KUKA KRL program: UP999.src, Up999.dat

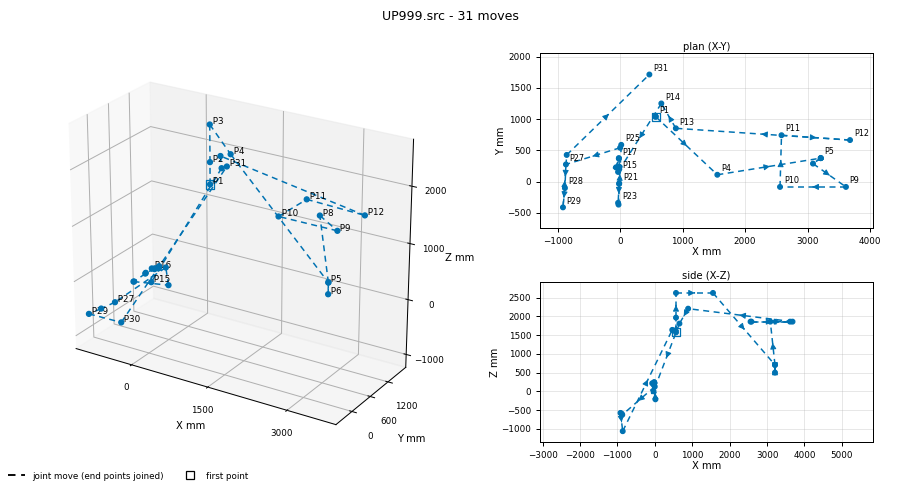
[picture p0: tool path of UP999.src, 31 of 31 moves have a stored position in this frame; points joined in program order, loops and branches not executed]
--- UP999.src ---
&ACCESS RVP2
&REL 75
&COMMENT israbiaoding
&PARAM EDITMASK = Up999[1-999]
&PARAM TPVW_VERSION = 8.3.17
&PARAM TEMPLATE = C:\KRC\Roboter\Template\upvorgabe
&PARAM DISKPATH = KRC:\R1\UPs
DEF UP999()
   ; FOLD UP Anfang;%{SE} %MKUKATPVW
   SPS_N=-1
   SPS_FERTIG=FALSE
   IF NOT CALLBYSELECT THEN
      INTERRUPT DECL 10 WHEN $CYCFLAG[254]==FALSE DO VW(#FB_STOP,TRUE)
      INTERRUPT ON 10
      INT10=TRUE
      VW_USR_R (#USR_INIT)
   ENDIF
   VW(#VW_INIT_UP,TRUE)
   ; ENDFOLD
   ;FOLD PTP VB=100% VE=0% ACC=100% RobWzg=0 Base=0 SPSTrig=0[1/100s]  ;%{P}%MKUKATPVW,%CMOVE8,%VPTP,%P 1:1, 2: VB=, 3:100, 4:%, 5: VE=, 6:0, 7:%, 8: ACC=, 9:100, 10:%, 11: RobWzg=, 12:0, 13: Base=, 14:0, 15: SPSTrig=, 16:0, 17:[1/100s], 18: , 19:1, 20:-1, 21:-1
      ;FOLD 1: ;%{SE}%MKUKATPVW
      ;ENDFOLD
      ;FOLD {H}
         VW_MPARA_ACT=P1_D
         Act_P1 = P1
         Act_P2 = P1
         VW(#MPARA,TRUE)
         PTP P1
         $ADVANCE=1
      ;ENDFOLD
   ;ENDFOLD
   ;FOLD PTP VB=100% VE=0% ACC=100% RobWzg=0 Base=0 SPSTrig=0[1/100s]  ;%{P}%MKUKATPVW,%CMOVE8,%VPTP,%P 1:1, 2: VB=, 3:100, 4:%, 5: VE=, 6:0, 7:%, 8: ACC=, 9:100, 10:%, 11: RobWzg=, 12:0, 13: Base=, 14:0, 15: SPSTrig=, 16:0, 17:[1/100s], 18: , 19:2, 20:-1, 21:-1
      ;FOLD 1: ;%{SE}%MKUKATPVW
      ;ENDFOLD
      ;FOLD {H}
         VW_MPARA_ACT=P2_D
         Act_P1 = P2
         Act_P2 = P2
         VW(#MPARA,TRUE)
         PTP P2
         $ADVANCE=1
      ;ENDFOLD
   ;ENDFOLD
   ;FOLD PTP VB=100% VE=0% ACC=100% RobWzg=0 Base=0 SPSTrig=0[1/100s]  ;%{P}%MKUKATPVW,%CMOVE8,%VPTP,%P 1:1, 2: VB=, 3:100, 4:%, 5: VE=, 6:0, 7:%, 8: ACC=, 9:100, 10:%, 11: RobWzg=, 12:0, 13: Base=, 14:0, 15: SPSTrig=, 16:0, 17:[1/100s], 18: , 19:3, 20:-1, 21:-1
      ;FOLD 1: ;%{SE}%MKUKATPVW
      ;ENDFOLD
      ;FOLD {H}
         VW_MPARA_ACT=P3_D
         Act_P1 = P3
         Act_P2 = P3
         VW(#MPARA,TRUE)
         PTP P3
         $ADVANCE=1
      ;ENDFOLD
   ;ENDFOLD
   ;FOLD PTP VB=100% VE=0% ACC=100% RobWzg=0 Base=0 SPSTrig=0[1/100s]  ;%{P}%MKUKATPVW,%CMOVE8,%VPTP,%P 1:1, 2: VB=, 3:100, 4:%, 5: VE=, 6:0, 7:%, 8: ACC=, 9:100, 10:%, 11: RobWzg=, 12:0, 13: Base=, 14:0, 15: SPSTrig=, 16:0, 17:[1/100s], 18: , 19:4, 20:-1, 21:-1
      ;FOLD 1: ;%{SE}%MKUKATPVW
      ;ENDFOLD
      ;FOLD {H}
         VW_MPARA_ACT=P4_D
         Act_P1 = P4
         Act_P2 = P4
         VW(#MPARA,TRUE)
         PTP P4
         $ADVANCE=1
      ;ENDFOLD
   ;ENDFOLD
   ;FOLD PTP VB=100% VE=0% ACC=100% RobWzg=21 Base=0 SPSTrig=0[1/100s]  ;%{P}%MKUKATPVW,%CMOVE8,%VPTP,%P 1:1, 2: VB=, 3:100, 4:%, 5: VE=, 6:0, 7:%, 8: ACC=, 9:100, 10:%, 11: RobWzg=, 12:21, 13: Base=, 14:0, 15: SPSTrig=, 16:0, 17:[1/100s], 18: , 19:5, 20:-1, 21:-1
      ;FOLD 1: ;%{SE}%MKUKATPVW
      ;ENDFOLD
      ;FOLD {H}
         VW_MPARA_ACT=P5_D
         Act_P1 = P5
         Act_P2 = P5
         VW(#MPARA,TRUE)
         PTP P5
         $ADVANCE=1
      ;ENDFOLD
   ;ENDFOLD
   ;FOLD -- zhongxintcp -- ;%{PSE}%MKUKATPVW,%CVW_COM,%VCOMMENT,%P 1:Comment:, 2:zhongxintcp
      ;FOLD {H}
         M_COMMENT("zhongxintcp")
      ;ENDFOLD
   ;ENDFOLD
   ;FOLD PTP VB=100% VE=0% ACC=100% RobWzg=21 Base=0 SPSTrig=0[1/100s]  ;%{P}%MKUKATPVW,%CMOVE8,%VPTP,%P 1:1, 2: VB=, 3:100, 4:%, 5: VE=, 6:0, 7:%, 8: ACC=, 9:100, 10:%, 11: RobWzg=, 12:21, 13: Base=, 14:0, 15: SPSTrig=, 16:0, 17:[1/100s], 18: , 19:6, 20:-1, 21:-1
      ;FOLD 1: ;%{SE}%MKUKATPVW
      ;ENDFOLD
      ;FOLD {H}
         VW_MPARA_ACT=P6_D
         Act_P1 = P6
         Act_P2 = P6
         VW(#MPARA,TRUE)
         PTP P6
         $ADVANCE=1
      ;ENDFOLD
   ;ENDFOLD
   ;FOLD PTP VB=100% VE=0% ACC=100% RobWzg=21 Base=0 SPSTrig=0[1/100s]  ;%{P}%MKUKATPVW,%CMOVE8,%VPTP,%P 1:1, 2: VB=, 3:100, 4:%, 5: VE=, 6:0, 7:%, 8: ACC=, 9:100, 10:%, 11: RobWzg=, 12:21, 13: Base=, 14:0, 15: SPSTrig=, 16:0, 17:[1/100s], 18: , 19:7, 20:-1, 21:-1
      ;FOLD 1: ;%{SE}%MKUKATPVW
      ;ENDFOLD
      ;FOLD {H}
         VW_MPARA_ACT=P7_D
         Act_P1 = P7
         Act_P2 = P7
         VW(#MPARA,TRUE)
         PTP P7
         $ADVANCE=1
      ;ENDFOLD
   ;ENDFOLD
   ;FOLD -- 1zhong -- ;%{PSE}%MKUKATPVW,%CVW_COM,%VCOMMENT,%P 1:Comment:, 2:1zhong
      ;FOLD {H}
         M_COMMENT("1zhong")
      ;ENDFOLD
   ;ENDFOLD
   ;FOLD PTP VB=100% VE=0% ACC=100% RobWzg=0 Base=0 SPSTrig=0[1/100s]  ;%{P}%MKUKATPVW,%CMOVE8,%VPTP,%P 1:1, 2: VB=, 3:100, 4:%, 5: VE=, 6:0, 7:%, 8: ACC=, 9:100, 10:%, 11: RobWzg=, 12:0, 13: Base=, 14:0, 15: SPSTrig=, 16:0, 17:[1/100s], 18: , 19:8, 20:-1, 21:-1
      ;FOLD 1: ;%{SE}%MKUKATPVW
      ;ENDFOLD
      ;FOLD {H}
         VW_MPARA_ACT=P8_D
         Act_P1 = P8
         Act_P2 = P8
         VW(#MPARA,TRUE)
         PTP P8
         $ADVANCE=1
      ;ENDFOLD
   ;ENDFOLD
   ;FOLD -- 2 -- ;%{PSE}%MKUKATPVW,%CVW_COM,%VCOMMENT,%P 1:Comment:, 2:2
      ;FOLD {H}
         M_COMMENT("2")
      ;ENDFOLD
   ;ENDFOLD
   ;FOLD PTP VB=100% VE=0% ACC=100% RobWzg=0 Base=0 SPSTrig=0[1/100s]  ;%{P}%MKUKATPVW,%CMOVE8,%VPTP,%P 1:1, 2: VB=, 3:100, 4:%, 5: VE=, 6:0, 7:%, 8: ACC=, 9:100, 10:%, 11: RobWzg=, 12:0, 13: Base=, 14:0, 15: SPSTrig=, 16:0, 17:[1/100s], 18: , 19:9, 20:-1, 21:-1
      ;FOLD 1: ;%{SE}%MKUKATPVW
      ;ENDFOLD
      ;FOLD {H}
         VW_MPARA_ACT=P9_D
         Act_P1 = P9
         Act_P2 = P9
         VW(#MPARA,TRUE)
         PTP P9
         $ADVANCE=1
      ;ENDFOLD
   ;ENDFOLD
   ;FOLD -- 3 -- ;%{PSE}%MKUKATPVW,%CVW_COM,%VCOMMENT,%P 1:Comment:, 2:3
      ;FOLD {H}
         M_COMMENT("3")
      ;ENDFOLD
   ;ENDFOLD
   ;FOLD PTP VB=100% VE=0% ACC=100% RobWzg=0 Base=0 SPSTrig=0[1/100s]  ;%{P}%MKUKATPVW,%CMOVE8,%VPTP,%P 1:1, 2: VB=, 3:100, 4:%, 5: VE=, 6:0, 7:%, 8: ACC=, 9:100, 10:%, 11: RobWzg=, 12:0, 13: Base=, 14:0, 15: SPSTrig=, 16:0, 17:[1/100s], 18: , 19:10, 20:-1, 21:-1
      ;FOLD 1: ;%{SE}%MKUKATPVW
      ;ENDFOLD
      ;FOLD {H}
         VW_MPARA_ACT=P10_D
         Act_P1 = P10
         Act_P2 = P10
         VW(#MPARA,TRUE)
         PTP P10
         $ADVANCE=1
      ;ENDFOLD
   ;ENDFOLD
   ;FOLD -- 4 -- ;%{PSE}%MKUKATPVW,%CVW_COM,%VCOMMENT,%P 1:Comment:, 2:4
      ;FOLD {H}
         M_COMMENT("4")
      ;ENDFOLD
   ;ENDFOLD
   ;FOLD PTP VB=100% VE=0% ACC=100% RobWzg=0 Base=0 SPSTrig=0[1/100s]  ;%{P}%MKUKATPVW,%CMOVE8,%VPTP,%P 1:1, 2: VB=, 3:100, 4:%, 5: VE=, 6:0, 7:%, 8: ACC=, 9:100, 10:%, 11: RobWzg=, 12:0, 13: Base=, 14:0, 15: SPSTrig=, 16:0, 17:[1/100s], 18: , 19:11, 20:-1, 21:-1
      ;FOLD 1: ;%{SE}%MKUKATPVW
      ;ENDFOLD
      ;FOLD {H}
         VW_MPARA_ACT=P11_D
         Act_P1 = P11
         Act_P2 = P11
         VW(#MPARA,TRUE)
         PTP P11
         $ADVANCE=1
      ;ENDFOLD
   ;ENDFOLD
   ;FOLD -- 5 -- ;%{PSE}%MKUKATPVW,%CVW_COM,%VCOMMENT,%P 1:Comment:, 2:5
      ;FOLD {H}
         M_COMMENT("5")
      ;ENDFOLD
   ;ENDFOLD
   ;FOLD PTP VB=100% VE=0% ACC=100% RobWzg=0 Base=0 SPSTrig=0[1/100s]  ;%{P}%MKUKATPVW,%CMOVE8,%VPTP,%P 1:1, 2: VB=, 3:100, 4:%, 5: VE=, 6:0, 7:%, 8: ACC=, 9:100, 10:%, 11: RobWzg=, 12:0, 13: Base=, 14:0, 15: SPSTrig=, 16:0, 17:[1/100s], 18: , 19:12, 20:-1, 21:-1
      ;FOLD 1: ;%{SE}%MKUKATPVW
      ;ENDFOLD
      ;FOLD {H}
         VW_MPARA_ACT=P12_D
         Act_P1 = P12
         Act_P2 = P12
         VW(#MPARA,TRUE)
         PTP P12
         $ADVANCE=1
      ;ENDFOLD
   ;ENDFOLD
   ;FOLD -- redian -- ;%{PSE}%MKUKATPVW,%CVW_COM,%VCOMMENT,%P 1:Comment:, 2:redian
      ;FOLD {H}
         M_COMMENT("redian")
      ;ENDFOLD
   ;ENDFOLD
   ;FOLD PTP VB=100% VE=0% ACC=100% RobWzg=0 Base=0 SPSTrig=0[1/100s]  ;%{P}%MKUKATPVW,%CMOVE8,%VPTP,%P 1:1, 2: VB=, 3:100, 4:%, 5: VE=, 6:0, 7:%, 8: ACC=, 9:100, 10:%, 11: RobWzg=, 12:0, 13: Base=, 14:0, 15: SPSTrig=, 16:0, 17:[1/100s], 18: , 19:13, 20:-1, 21:-1
      ;FOLD 1: ;%{SE}%MKUKATPVW
      ;ENDFOLD
      ;FOLD {H}
         VW_MPARA_ACT=P13_D
         Act_P1 = P13
         Act_P2 = P13
         VW(#MPARA,TRUE)
         PTP P13
         $ADVANCE=1
      ;ENDFOLD
   ;ENDFOLD
   ;FOLD PTP VB=100% VE=0% ACC=100% RobWzg=0 Base=0 SPSTrig=0[1/100s]  ;%{P}%MKUKATPVW,%CMOVE8,%VPTP,%P 1:1, 2: VB=, 3:100, 4:%, 5: VE=, 6:0, 7:%, 8: ACC=, 9:100, 10:%, 11: RobWzg=, 12:0, 13: Base=, 14:0, 15: SPSTrig=, 16:0, 17:[1/100s], 18: , 19:14, 20:-1, 21:-1
      ;FOLD 1: ;%{SE}%MKUKATPVW
      ;ENDFOLD
      ;FOLD {H}
         VW_MPARA_ACT=P14_D
         Act_P1 = P14
         Act_P2 = P14
         VW(#MPARA,TRUE)
         PTP P14
         $ADVANCE=1
      ;ENDFOLD
   ;ENDFOLD
   ;FOLD PTP VB=100% VE=0% ACC=100% RobWzg=21 Base=21 SPSTrig=0[1/100s]  ;%{P}%MKUKATPVW,%CMOVE8,%VPTP,%P 1:1, 2: VB=, 3:100, 4:%, 5: VE=, 6:0, 7:%, 8: ACC=, 9:100, 10:%, 11: RobWzg=, 12:21, 13: Base=, 14:21, 15: SPSTrig=, 16:0, 17:[1/100s], 18: , 19:15, 20:-1, 21:-1
      ;FOLD 1: ;%{SE}%MKUKATPVW
      ;ENDFOLD
      ;FOLD {H}
         VW_MPARA_ACT=P15_D
         Act_P1 = P15
         Act_P2 = P15
         VW(#MPARA,TRUE)
         PTP P15
         $ADVANCE=1
      ;ENDFOLD
   ;ENDFOLD
   ;FOLD PTP VB=100% VE=0% ACC=100% RobWzg=21 Base=21 SPSTrig=0[1/100s]  ;%{P}%MKUKATPVW,%CMOVE8,%VPTP,%P 1:1, 2: VB=, 3:100, 4:%, 5: VE=, 6:0, 7:%, 8: ACC=, 9:100, 10:%, 11: RobWzg=, 12:21, 13: Base=, 14:21, 15: SPSTrig=, 16:0, 17:[1/100s], 18: , 19:16, 20:-1, 21:-1
      ;FOLD 1: ;%{SE}%MKUKATPVW
      ;ENDFOLD
      ;FOLD {H}
         VW_MPARA_ACT=P16_D
         Act_P1 = P16
         Act_P2 = P16
         VW(#MPARA,TRUE)
         PTP P16
         $ADVANCE=1
      ;ENDFOLD
   ;ENDFOLD
   ;FOLD -- 1zs -- ;%{PSE}%MKUKATPVW,%CVW_COM,%VCOMMENT,%P 1:Comment:, 2:1zs
      ;FOLD {H}
         M_COMMENT("1zs")
      ;ENDFOLD
   ;ENDFOLD
   ;FOLD PTP VB=100% VE=0% ACC=100% RobWzg=21 Base=21 SPSTrig=0[1/100s]  ;%{P}%MKUKATPVW,%CMOVE8,%VPTP,%P 1:1, 2: VB=, 3:100, 4:%, 5: VE=, 6:0, 7:%, 8: ACC=, 9:100, 10:%, 11: RobWzg=, 12:21, 13: Base=, 14:21, 15: SPSTrig=, 16:0, 17:[1/100s], 18: , 19:17, 20:-1, 21:-1
      ;FOLD 1: ;%{SE}%MKUKATPVW
      ;ENDFOLD
      ;FOLD {H}
         VW_MPARA_ACT=P17_D
         Act_P1 = P17
         Act_P2 = P17
         VW(#MPARA,TRUE)
         PTP P17
         $ADVANCE=1
      ;ENDFOLD
   ;ENDFOLD
   ;FOLD PTP VB=100% VE=0% ACC=100% RobWzg=21 Base=21 SPSTrig=0[1/100s]  ;%{P}%MKUKATPVW,%CMOVE8,%VPTP,%P 1:1, 2: VB=, 3:100, 4:%, 5: VE=, 6:0, 7:%, 8: ACC=, 9:100, 10:%, 11: RobWzg=, 12:21, 13: Base=, 14:21, 15: SPSTrig=, 16:0, 17:[1/100s], 18: , 19:18, 20:-1, 21:-1
      ;FOLD 1: ;%{SE}%MKUKATPVW
      ;ENDFOLD
      ;FOLD {H}
         VW_MPARA_ACT=P18_D
         Act_P1 = P18
         Act_P2 = P18
         VW(#MPARA,TRUE)
         PTP P18
         $ADVANCE=1
      ;ENDFOLD
   ;ENDFOLD
   ;FOLD -- 2ys -- ;%{PSE}%MKUKATPVW,%CVW_COM,%VCOMMENT,%P 1:Comment:, 2:2ys
      ;FOLD {H}
         M_COMMENT("2ys")
      ;ENDFOLD
   ;ENDFOLD
   ;FOLD PTP VB=100% VE=0% ACC=100% RobWzg=21 Base=21 SPSTrig=0[1/100s]  ;%{P}%MKUKATPVW,%CMOVE8,%VPTP,%P 1:1, 2: VB=, 3:100, 4:%, 5: VE=, 6:0, 7:%, 8: ACC=, 9:100, 10:%, 11: RobWzg=, 12:21, 13: Base=, 14:21, 15: SPSTrig=, 16:0, 17:[1/100s], 18: , 19:19, 20:-1, 21:-1
      ;FOLD 1: ;%{SE}%MKUKATPVW
      ;ENDFOLD
      ;FOLD {H}
         VW_MPARA_ACT=P19_D
         Act_P1 = P19
         Act_P2 = P19
         VW(#MPARA,TRUE)
         PTP P19
         $ADVANCE=1
      ;ENDFOLD
   ;ENDFOLD
   ;FOLD PTP VB=100% VE=0% ACC=100% RobWzg=21 Base=21 SPSTrig=0[1/100s]  ;%{P}%MKUKATPVW,%CMOVE8,%VPTP,%P 1:1, 2: VB=, 3:100, 4:%, 5: VE=, 6:0, 7:%, 8: ACC=, 9:100, 10:%, 11: RobWzg=, 12:21, 13: Base=, 14:21, 15: SPSTrig=, 16:0, 17:[1/100s], 18: , 19:20, 20:-1, 21:-1
      ;FOLD 1: ;%{SE}%MKUKATPVW
      ;ENDFOLD
      ;FOLD {H}
         VW_MPARA_ACT=P20_D
         Act_P1 = P20
         Act_P2 = P20
         VW(#MPARA,TRUE)
         PTP P20
         $ADVANCE=1
      ;ENDFOLD
   ;ENDFOLD
   ;FOLD -- 3zx -- ;%{PSE}%MKUKATPVW,%CVW_COM,%VCOMMENT,%P 1:Comment:, 2:3zx
      ;FOLD {H}
         M_COMMENT("3zx")
      ;ENDFOLD
   ;ENDFOLD
   ;FOLD PTP VB=100% VE=0% ACC=100% RobWzg=21 Base=21 SPSTrig=0[1/100s]  ;%{P}%MKUKATPVW,%CMOVE8,%VPTP,%P 1:1, 2: VB=, 3:100, 4:%, 5: VE=, 6:0, 7:%, 8: ACC=, 9:100, 10:%, 11: RobWzg=, 12:21, 13: Base=, 14:21, 15: SPSTrig=, 16:0, 17:[1/100s], 18: , 19:21, 20:-1, 21:-1
      ;FOLD 1: ;%{SE}%MKUKATPVW
      ;ENDFOLD
      ;FOLD {H}
         VW_MPARA_ACT=P21_D
         Act_P1 = P21
         Act_P2 = P21
         VW(#MPARA,TRUE)
         PTP P21
         $ADVANCE=1
      ;ENDFOLD
   ;ENDFOLD
   ;FOLD PTP VB=100% VE=0% ACC=100% RobWzg=21 Base=21 SPSTrig=5[1/100s]  ;%{P}%MKUKATPVW,%CMOVE8,%VPTP,%P 1:1, 2: VB=, 3:100, 4:%, 5: VE=, 6:0, 7:%, 8: ACC=, 9:100, 10:%, 11: RobWzg=, 12:21, 13: Base=, 14:21, 15: SPSTrig=, 16:5, 17:[1/100s], 18: , 19:22, 20:-1, 21:-1
      ;FOLD 1: ;%{SE}%MKUKATPVW
      ;ENDFOLD
      ;FOLD {H}
         VW_MPARA_ACT=P22_D
         Act_P1 = P22
         Act_P2 = P22
         VW(#MPARA,TRUE)
         PTP P22
         $ADVANCE=1
      ;ENDFOLD
   ;ENDFOLD
   ;FOLD -- 4zz -- ;%{PSE}%MKUKATPVW,%CVW_COM,%VCOMMENT,%P 1:Comment:, 2:4zz
      ;FOLD {H}
         M_COMMENT("4zz")
      ;ENDFOLD
   ;ENDFOLD
   ;FOLD PTP VB=100% VE=0% ACC=100% RobWzg=21 Base=21 SPSTrig=0[1/100s]  ;%{P}%MKUKATPVW,%CMOVE8,%VPTP,%P 1:1, 2: VB=, 3:100, 4:%, 5: VE=, 6:0, 7:%, 8: ACC=, 9:100, 10:%, 11: RobWzg=, 12:21, 13: Base=, 14:21, 15: SPSTrig=, 16:0, 17:[1/100s], 18: , 19:23, 20:-1, 21:-1
      ;FOLD 1: ;%{SE}%MKUKATPVW
      ;ENDFOLD
      ;FOLD {H}
         VW_MPARA_ACT=P23_D
         Act_P1 = P23
         Act_P2 = P23
         VW(#MPARA,TRUE)
         PTP P23
         $ADVANCE=1
      ;ENDFOLD
   ;ENDFOLD
   ;FOLD -- 4 -- ;%{PSE}%MKUKATPVW,%CVW_COM,%VCOMMENT,%P 1:Comment:, 2:4
      ;FOLD {H}
         M_COMMENT("4")
      ;ENDFOLD
   ;ENDFOLD
   ;FOLD PTP VB=100% VE=0% ACC=100% RobWzg=21 Base=21 SPSTrig=0[1/100s]  ;%{P}%MKUKATPVW,%CMOVE8,%VPTP,%P 1:1, 2: VB=, 3:100, 4:%, 5: VE=, 6:0, 7:%, 8: ACC=, 9:100, 10:%, 11: RobWzg=, 12:21, 13: Base=, 14:21, 15: SPSTrig=, 16:0, 17:[1/100s], 18: , 19:24, 20:-1, 21:-1
      ;FOLD 1: ;%{SE}%MKUKATPVW
      ;ENDFOLD
      ;FOLD {H}
         VW_MPARA_ACT=P24_D
         Act_P1 = P24
         Act_P2 = P24
         VW(#MPARA,TRUE)
         PTP P24
         $ADVANCE=1
      ;ENDFOLD
   ;ENDFOLD
   ;FOLD -- 3 -- ;%{PSE}%MKUKATPVW,%CVW_COM,%VCOMMENT,%P 1:Comment:, 2:3
      ;FOLD {H}
         M_COMMENT("3")
      ;ENDFOLD
   ;ENDFOLD
   ;FOLD PTP VB=100% VE=0% ACC=100% RobWzg=21 Base=21 SPSTrig=0[1/100s]  ;%{P}%MKUKATPVW,%CMOVE8,%VPTP,%P 1:1, 2: VB=, 3:100, 4:%, 5: VE=, 6:0, 7:%, 8: ACC=, 9:100, 10:%, 11: RobWzg=, 12:21, 13: Base=, 14:21, 15: SPSTrig=, 16:0, 17:[1/100s], 18: , 19:25, 20:-1, 21:-1
      ;FOLD 1: ;%{SE}%MKUKATPVW
      ;ENDFOLD
      ;FOLD {H}
         VW_MPARA_ACT=P25_D
         Act_P1 = P25
         Act_P2 = P25
         VW(#MPARA,TRUE)
         PTP P25
         $ADVANCE=1
      ;ENDFOLD
   ;ENDFOLD
   ;FOLD -- 33 -- ;%{PSE}%MKUKATPVW,%CVW_COM,%VCOMMENT,%P 1:Comment:, 2:33
      ;FOLD {H}
         M_COMMENT("33")
      ;ENDFOLD
   ;ENDFOLD
   ;FOLD PTP VB=100% VE=0% ACC=100% RobWzg=21 Base=21 SPSTrig=0[1/100s]  ;%{P}%MKUKATPVW,%CMOVE8,%VPTP,%P 1:1, 2: VB=, 3:100, 4:%, 5: VE=, 6:0, 7:%, 8: ACC=, 9:100, 10:%, 11: RobWzg=, 12:21, 13: Base=, 14:21, 15: SPSTrig=, 16:0, 17:[1/100s], 18: , 19:26, 20:-1, 21:-1
      ;FOLD 1: ;%{SE}%MKUKATPVW
      ;ENDFOLD
      ;FOLD {H}
         VW_MPARA_ACT=P26_D
         Act_P1 = P26
         Act_P2 = P26
         VW(#MPARA,TRUE)
         PTP P26
         $ADVANCE=1
      ;ENDFOLD
   ;ENDFOLD
   ;FOLD -- 1 -- ;%{PSE}%MKUKATPVW,%CVW_COM,%VCOMMENT,%P 1:Comment:, 2:1
      ;FOLD {H}
         M_COMMENT("1")
      ;ENDFOLD
   ;ENDFOLD
   ;FOLD PTP VB=100% VE=0% ACC=100% RobWzg=21 Base=21 SPSTrig=0[1/100s]  ;%{P}%MKUKATPVW,%CMOVE8,%VPTP,%P 1:1, 2: VB=, 3:100, 4:%, 5: VE=, 6:0, 7:%, 8: ACC=, 9:100, 10:%, 11: RobWzg=, 12:21, 13: Base=, 14:21, 15: SPSTrig=, 16:0, 17:[1/100s], 18: , 19:27, 20:-1, 21:-1
      ;FOLD 1: ;%{SE}%MKUKATPVW
      ;ENDFOLD
      ;FOLD {H}
         VW_MPARA_ACT=P27_D
         Act_P1 = P27
         Act_P2 = P27
         VW(#MPARA,TRUE)
         PTP P27
         $ADVANCE=1
      ;ENDFOLD
   ;ENDFOLD
   ;FOLD -- 2 -- ;%{PSE}%MKUKATPVW,%CVW_COM,%VCOMMENT,%P 1:Comment:, 2:2
      ;FOLD {H}
         M_COMMENT("2")
      ;ENDFOLD
   ;ENDFOLD
   ;FOLD PTP VB=100% VE=0% ACC=100% RobWzg=21 Base=21 SPSTrig=0[1/100s]  ;%{P}%MKUKATPVW,%CMOVE8,%VPTP,%P 1:1, 2: VB=, 3:100, 4:%, 5: VE=, 6:0, 7:%, 8: ACC=, 9:100, 10:%, 11: RobWzg=, 12:21, 13: Base=, 14:21, 15: SPSTrig=, 16:0, 17:[1/100s], 18: , 19:28, 20:-1, 21:-1
      ;FOLD 1: ;%{SE}%MKUKATPVW
      ;ENDFOLD
      ;FOLD {H}
         VW_MPARA_ACT=P28_D
         Act_P1 = P28
         Act_P2 = P28
         VW(#MPARA,TRUE)
         PTP P28
         $ADVANCE=1
      ;ENDFOLD
   ;ENDFOLD
   ;FOLD -- 3 -- ;%{PSE}%MKUKATPVW,%CVW_COM,%VCOMMENT,%P 1:Comment:, 2:3
      ;FOLD {H}
         M_COMMENT("3")
      ;ENDFOLD
   ;ENDFOLD
   ;FOLD PTP VB=100% VE=0% ACC=100% RobWzg=21 Base=21 SPSTrig=0[1/100s]  ;%{P}%MKUKATPVW,%CMOVE8,%VPTP,%P 1:1, 2: VB=, 3:100, 4:%, 5: VE=, 6:0, 7:%, 8: ACC=, 9:100, 10:%, 11: RobWzg=, 12:21, 13: Base=, 14:21, 15: SPSTrig=, 16:0, 17:[1/100s], 18: , 19:29, 20:-1, 21:-1
      ;FOLD 1: ;%{SE}%MKUKATPVW
      ;ENDFOLD
      ;FOLD {H}
         VW_MPARA_ACT=P29_D
         Act_P1 = P29
         Act_P2 = P29
         VW(#MPARA,TRUE)
         PTP P29
         $ADVANCE=1
      ;ENDFOLD
   ;ENDFOLD
   ;FOLD -- 4 -- ;%{PSE}%MKUKATPVW,%CVW_COM,%VCOMMENT,%P 1:Comment:, 2:4
      ;FOLD {H}
         M_COMMENT("4")
      ;ENDFOLD
   ;ENDFOLD
   ;FOLD PTP VB=100% VE=0% ACC=100% RobWzg=21 Base=21 SPSTrig=0[1/100s]  ;%{P}%MKUKATPVW,%CMOVE8,%VPTP,%P 1:1, 2: VB=, 3:100, 4:%, 5: VE=, 6:0, 7:%, 8: ACC=, 9:100, 10:%, 11: RobWzg=, 12:21, 13: Base=, 14:21, 15: SPSTrig=, 16:0, 17:[1/100s], 18: , 19:30, 20:-1, 21:-1
      ;FOLD 1: ;%{SE}%MKUKATPVW
      ;ENDFOLD
      ;FOLD {H}
         VW_MPARA_ACT=P30_D
         Act_P1 = P30
         Act_P2 = P30
         VW(#MPARA,TRUE)
         PTP P30
         $ADVANCE=1
      ;ENDFOLD
   ;ENDFOLD
   ;FOLD PTP VB=100% VE=0% ACC=100% RobWzg=0 Base=0 SPSTrig=0[1/100s]  ;%{P}%MKUKATPVW,%CMOVE8,%VPTP,%P 1:1, 2: VB=, 3:100, 4:%, 5: VE=, 6:0, 7:%, 8: ACC=, 9:100, 10:%, 11: RobWzg=, 12:0, 13: Base=, 14:0, 15: SPSTrig=, 16:0, 17:[1/100s], 18: , 19:31, 20:-1, 21:-1
      ;FOLD 1: ;%{SE}%MKUKATPVW
      ;ENDFOLD
      ;FOLD {H}
         VW_MPARA_ACT=P31_D
         Act_P1 = P31
         Act_P2 = P31
         VW(#MPARA,TRUE)
         PTP P31
         $ADVANCE=1
      ;ENDFOLD
   ;ENDFOLD
   ; FOLD ;%{H}
END
DEF SPS_TRIG(NO :IN)
   INT NO
   INT VW_STOP
   BOOL UES
   BOOL ANA_UES
   BOOL ANA_TRIG
   VW_STOP=$VW_PSPS_STOP
   UES=FALSE
   ANA_UES=FALSE
   ANA_TRIG=FALSE
   IF ((NO>10000) AND (NO<20000)) THEN
      NO=NO-10000
      UES=TRUE
   ENDIF
   IF ((NO>20000) AND (NO<30000)) THEN
      NO=NO-20000
      ANA_TRIG=TRUE
   ENDIF
   IF NO>30000 THEN
      NO=NO-30000
      ANA_UES=TRUE
      ANA_TRIG=TRUE
   ENDIF
   ; FOLD ;%{H}
   IF ((VW_STOP B_AND 'B0001') > 0) THEN
      ;-- Trigger vorzeitig geschaltet (delay < 0) oder MStep
      IF (((VW_STOP B_AND 'B0110') > 0) AND ($MODE_OP<>#EX)) THEN
         ;-- MStep oder BCO Bewegung
         HALT
      ENDIF
   ENDIF
   ; ENDFOLD
   IF (SEARCH_END) THEN
      SEARCH_END = FALSE
      INTERRUPT OFF 39
   ENDIF
   SWITCH NO
      CASE 1
         ;FOLD SPS_TRIG1 {H}
         ;ENDFOLD
      CASE 2
         ;FOLD SPS_TRIG2 {H}
         ;ENDFOLD
      CASE 3
         ;FOLD SPS_TRIG3 {H}
         ;ENDFOLD
      CASE 4
         ;FOLD SPS_TRIG4 {H}
         ;ENDFOLD
      CASE 5
         ;FOLD SPS_TRIG5 {H}
         ;ENDFOLD
      CASE 6
         ;FOLD SPS_TRIG6 {H}
         ;ENDFOLD
      CASE 7
         ;FOLD SPS_TRIG7 {H}
         ;ENDFOLD
      CASE 8
         ;FOLD SPS_TRIG8 {H}
         ;ENDFOLD
      CASE 9
         ;FOLD SPS_TRIG9 {H}
         ;ENDFOLD
      CASE 10
         ;FOLD SPS_TRIG10 {H}
         ;ENDFOLD
      CASE 11
         ;FOLD SPS_TRIG11 {H}
         ;ENDFOLD
      CASE 12
         ;FOLD SPS_TRIG12 {H}
         ;ENDFOLD
      CASE 13
         ;FOLD SPS_TRIG13 {H}
         ;ENDFOLD
      CASE 14
         ;FOLD SPS_TRIG14 {H}
         ;ENDFOLD
      CASE 15
         ;FOLD SPS_TRIG15 {H}
         ;ENDFOLD
      CASE 16
         ;FOLD SPS_TRIG16 {H}
         ;ENDFOLD
      CASE 17
         ;FOLD SPS_TRIG17 {H}
         ;ENDFOLD
      CASE 18
         ;FOLD SPS_TRIG18 {H}
         ;ENDFOLD
      CASE 19
         ;FOLD SPS_TRIG19 {H}
         ;ENDFOLD
      CASE 20
         ;FOLD SPS_TRIG20 {H}
         ;ENDFOLD
      CASE 21
         ;FOLD SPS_TRIG21 {H}
         ;ENDFOLD
      CASE 22
         ;FOLD SPS_TRIG22 {H}
         ;ENDFOLD
      CASE 23
         ;FOLD SPS_TRIG23 {H}
         ;ENDFOLD
      CASE 24
         ;FOLD SPS_TRIG24 {H}
         ;ENDFOLD
      CASE 25
         ;FOLD SPS_TRIG25 {H}
         ;ENDFOLD
      CASE 26
         ;FOLD SPS_TRIG26 {H}
         ;ENDFOLD
      CASE 27
         ;FOLD SPS_TRIG27 {H}
         ;ENDFOLD
      CASE 28
         ;FOLD SPS_TRIG28 {H}
         ;ENDFOLD
      CASE 29
         ;FOLD SPS_TRIG29 {H}
         ;ENDFOLD
      CASE 30
         ;FOLD SPS_TRIG30 {H}
         ;ENDFOLD
      CASE 31
         ;FOLD SPS_TRIG31 {H}
         ;ENDFOLD
      CASE 32
         ;FOLD SPS_TRIG32 {H}
         ;ENDFOLD
      CASE 33
         ;FOLD SPS_TRIG33 {H}
         ;ENDFOLD
      CASE 34
         ;FOLD SPS_TRIG34 {H}
         ;ENDFOLD
      CASE 35
         ;FOLD SPS_TRIG35 {H}
         ;ENDFOLD
      CASE 36
         ;FOLD SPS_TRIG36 {H}
         ;ENDFOLD
      CASE 37
         ;FOLD SPS_TRIG37 {H}
         ;ENDFOLD
      CASE 38
         ;FOLD SPS_TRIG38 {H}
         ;ENDFOLD
      CASE 39
         ;FOLD SPS_TRIG39 {H}
         ;ENDFOLD
      CASE 40
         ;FOLD SPS_TRIG40 {H}
         ;ENDFOLD
      CASE 41
         ;FOLD SPS_TRIG41 {H}
         ;ENDFOLD
      CASE 42
         ;FOLD SPS_TRIG42 {H}
         ;ENDFOLD
      CASE 43
         ;FOLD SPS_TRIG43 {H}
         ;ENDFOLD
      CASE 44
         ;FOLD SPS_TRIG44 {H}
         ;ENDFOLD
      CASE 45
         ;FOLD SPS_TRIG45 {H}
         ;ENDFOLD
      CASE 46
         ;FOLD SPS_TRIG46 {H}
         ;ENDFOLD
      CASE 47
         ;FOLD SPS_TRIG47 {H}
         ;ENDFOLD
      CASE 48
         ;FOLD SPS_TRIG48 {H}
         ;ENDFOLD
      CASE 49
         ;FOLD SPS_TRIG49 {H}
         ;ENDFOLD
      CASE 50
         ;FOLD SPS_TRIG50 {H}
         ;ENDFOLD
      CASE 51
         ;FOLD SPS_TRIG51 {H}
         ;ENDFOLD
      CASE 52
         ;FOLD SPS_TRIG52 {H}
         ;ENDFOLD
      CASE 53
         ;FOLD SPS_TRIG53 {H}
         ;ENDFOLD
      CASE 54
         ;FOLD SPS_TRIG54 {H}
         ;ENDFOLD
      CASE 55
         ;FOLD SPS_TRIG55 {H}
         ;ENDFOLD
      CASE 56
         ;FOLD SPS_TRIG56 {H}
         ;ENDFOLD
      CASE 57
         ;FOLD SPS_TRIG57 {H}
         ;ENDFOLD
      CASE 58
         ;FOLD SPS_TRIG58 {H}
         ;ENDFOLD
      CASE 59
         ;FOLD SPS_TRIG59 {H}
         ;ENDFOLD
      CASE 60
         ;FOLD SPS_TRIG60 {H}
         ;ENDFOLD
      CASE 61
         ;FOLD SPS_TRIG61 {H}
         ;ENDFOLD
      CASE 62
         ;FOLD SPS_TRIG62 {H}
         ;ENDFOLD
      CASE 63
         ;FOLD SPS_TRIG63 {H}
         ;ENDFOLD
      CASE 64
         ;FOLD SPS_TRIG64 {H}
         ;ENDFOLD
      CASE 65
         ;FOLD SPS_TRIG65 {H}
         ;ENDFOLD
      CASE 66
         ;FOLD SPS_TRIG66 {H}
         ;ENDFOLD
      CASE 67
         ;FOLD SPS_TRIG67 {H}
         ;ENDFOLD
      CASE 68
         ;FOLD SPS_TRIG68 {H}
         ;ENDFOLD
      CASE 69
         ;FOLD SPS_TRIG69 {H}
         ;ENDFOLD
      CASE 70
         ;FOLD SPS_TRIG70 {H}
         ;ENDFOLD
      CASE 71
         ;FOLD SPS_TRIG71 {H}
         ;ENDFOLD
      CASE 72
         ;FOLD SPS_TRIG72 {H}
         ;ENDFOLD
      CASE 73
         ;FOLD SPS_TRIG73 {H}
         ;ENDFOLD
      CASE 74
         ;FOLD SPS_TRIG74 {H}
         ;ENDFOLD
      CASE 75
         ;FOLD SPS_TRIG75 {H}
         ;ENDFOLD
      CASE 76
         ;FOLD SPS_TRIG76 {H}
         ;ENDFOLD
      CASE 77
         ;FOLD SPS_TRIG77 {H}
         ;ENDFOLD
      CASE 78
         ;FOLD SPS_TRIG78 {H}
         ;ENDFOLD
      CASE 79
         ;FOLD SPS_TRIG79 {H}
         ;ENDFOLD
      CASE 80
         ;FOLD SPS_TRIG80 {H}
         ;ENDFOLD
      CASE 81
         ;FOLD SPS_TRIG81 {H}
         ;ENDFOLD
      CASE 82
         ;FOLD SPS_TRIG82 {H}
         ;ENDFOLD
      CASE 83
         ;FOLD SPS_TRIG83 {H}
         ;ENDFOLD
      CASE 84
         ;FOLD SPS_TRIG84 {H}
         ;ENDFOLD
      CASE 85
         ;FOLD SPS_TRIG85 {H}
         ;ENDFOLD
      CASE 86
         ;FOLD SPS_TRIG86 {H}
         ;ENDFOLD
      CASE 87
         ;FOLD SPS_TRIG87 {H}
         ;ENDFOLD
      CASE 88
         ;FOLD SPS_TRIG88 {H}
         ;ENDFOLD
      CASE 89
         ;FOLD SPS_TRIG89 {H}
         ;ENDFOLD
      CASE 90
         ;FOLD SPS_TRIG90 {H}
         ;ENDFOLD
      CASE 91
         ;FOLD SPS_TRIG91 {H}
         ;ENDFOLD
      CASE 92
         ;FOLD SPS_TRIG92 {H}
         ;ENDFOLD
      CASE 93
         ;FOLD SPS_TRIG93 {H}
         ;ENDFOLD
      CASE 94
         ;FOLD SPS_TRIG94 {H}
         ;ENDFOLD
      CASE 95
         ;FOLD SPS_TRIG95 {H}
         ;ENDFOLD
      CASE 96
         ;FOLD SPS_TRIG96 {H}
         ;ENDFOLD
      CASE 97
         ;FOLD SPS_TRIG97 {H}
         ;ENDFOLD
      CASE 98
         ;FOLD SPS_TRIG98 {H}
         ;ENDFOLD
      CASE 99
         ;FOLD SPS_TRIG99 {H}
         ;ENDFOLD
      CASE 100
         ;FOLD SPS_TRIG100 {H}
         ;ENDFOLD
      CASE 101
         ;FOLD SPS_TRIG101 {H}
         ;ENDFOLD
   DEFAULT
   ENDSWITCH
   ; FOLD ;%{H}
   IF ($MODE_OP<>#EX) THEN
      ;-- Trigger erst nach Wiederanstart geschaltet --
      IF ((((VW_STOP B_AND 'B10010') >0) AND ((VW_STOP B_AND 'B0001')<=0))) THEN
         ;-- MStep Bewegung --
         HALT
      ENDIF
   ENDIF
   ; ENDFOLD
   IF (NOT UES AND NOT ANA_TRIG) THEN
      SPS_FERTIG=TRUE
   ENDIF
   IF (NOT ANA_UES AND ANA_TRIG) THEN
      SPS_FERTIG_ANA=TRUE
   ENDIF
END
; ENDFOLD

--- Up999.dat ---
&ACCESS RVP2
&REL 75
&COMMENT israbiaoding
&PARAM EDITMASK = Up999[1-999]
&PARAM TPVW_VERSION = 8.3.17
&PARAM TEMPLATE = C:\KRC\Roboter\Template\upvorgabe
&PARAM DISKPATH = KRC:\R1\UPs
DEFDAT  Up999
; FOLD ;%{H} %MKUKATPVW
; ENDFOLD
; interface to basic routines
EXT  BAS (BAS_COMMAND  :IN,REAL  :IN )
; interface to VW-standard routines
EXT  VW (VW_COMMAND  :IN,BOOL  :IN,REAL  :IN,REAL  :IN,REAL  :IN,REAL  :IN,BOOL  :IN,E6POS  :IN )
; interface to VW_USER - Call
EXT  VW_USER (VW_USER_CMD  :IN,INT  :IN,REAL  :IN,REAL  :IN,REAL  :IN,REAL  :IN,REAL  :IN,REAL  :IN,REAL  :IN,REAL  :IN,REAL  :IN,BOOL  :IN )
EXT  VW_USR_R (VW_USER_CMD  :IN,INT  :IN,REAL  :IN,REAL  :IN,REAL  :IN,REAL  :IN,REAL  :IN,REAL  :IN,REAL  :IN,REAL  :IN,REAL  :IN,BOOL  :IN )
EXT  IBGN (IBGN_COMMAND  :IN,BOOL  :IN,REAL  :IN,REAL  :IN,BOOL  :IN,E6POS  :OUT )
; interface select routine
EXTFCT  INT  SELECT(SUBTYPE  :IN,INT  :IN,BOOL  :IN,ARI_TYP  :IN,INT  :IN,BOOL_TYP  :IN,INT  :IN,BOOL  :IN)
INT VW_NEXT_FREE=32
INT VW_NFREE_SPS=1
INT VW_MAX_SPS=101
DECL VW_MPARA_TYP P1_D={TOOL_NO 0,BASE_NO 0,VB 100,VE 0,ACC 100,TRG_TIME 0,MOVE_TYPE #PTP_MOTION}
DECL E6POS P1={X 566.159,Y 1040.67896,Z 1575.40503,A 52.8831787,B -10.8393602,C -173.993805,S 2,T 3,E1 -518.843384,E2 0.0,E3 0.0,E4 0.0,E5 0.0,E6 0.0}
DECL VW_MPARA_TYP P2_D={TOOL_NO 0,BASE_NO 0,VB 100,VE 0,ACC 100,TRG_TIME 0,MOVE_TYPE #PTP_MOTION}
DECL E6POS P2={X 566.159,Y 1040.67896,Z 1969.88599,A 56.1079712,B 78.1039276,C -113.386803,S 2,T 11,E1 -518.843384,E2 0.0,E3 0.0,E4 0.0,E5 0.0,E6 0.0}
DECL VW_MPARA_TYP P3_D={TOOL_NO 0,BASE_NO 0,VB 100,VE 0,ACC 100,TRG_TIME 0,MOVE_TYPE #PTP_MOTION}
DECL E6POS P3={X 566.159,Y 1040.67896,Z 2629.29395,A 56.1079712,B 78.1039276,C -113.386803,S 2,T 11,E1 -518.843384,E2 0.0,E3 0.0,E4 0.0,E5 0.0,E6 0.0}
DECL VW_MPARA_TYP P4_D={TOOL_NO 0,BASE_NO 0,VB 100,VE 0,ACC 100,TRG_TIME 0,MOVE_TYPE #PTP_MOTION}
DECL E6POS P4={X 1554.89905,Y 108.819801,Z 2629.29395,A -25.2928505,B 78.1039276,C -113.386803,S 2,T 10,E1 -518.843384,E2 0.0,E3 0.0,E4 0.0,E5 0.0,E6 0.0}
DECL VW_MPARA_TYP P5_D={TOOL_NO 21,BASE_NO 0,VB 100,VE 0,ACC 100,TRG_TIME 0,MOVE_TYPE #PTP_MOTION}
DECL E6POS P5={X 3211.20093,Y 374.839386,Z 706.640,A -82.5392,B -4.08844709,C -176.631,S 2,T 3,E1 -1250.45300,E2 0.0,E3 0.0,E4 0.0,E5 0.0,E6 0.0}
DECL VW_MPARA_TYP P6_D={TOOL_NO 21,BASE_NO 0,VB 100,VE 0,ACC 100,TRG_TIME 0,MOVE_TYPE #PTP_MOTION}
DECL E6POS P6={X 3211.20093,Y 374.839386,Z 501.234497,A -82.5392,B -4.08844709,C -176.631,S 2,T 3,E1 -1250.45300,E2 0.0,E3 0.0,E4 0.0,E5 0.0,E6 0.0}
DECL VW_MPARA_TYP P7_D={TOOL_NO 21,BASE_NO 0,VB 100,VE 0,ACC 100,TRG_TIME 0,MOVE_TYPE #PTP_MOTION}
DECL E6POS P7={X 3211.20093,Y 374.839294,Z 706.640,A -82.5392,B -4.08844709,C -176.631,S 2,T 3,E1 -1250.45300,E2 0.0,E3 0.0,E4 0.0,E5 0.0,E6 0.0}
DECL VW_MPARA_TYP P8_D={TOOL_NO 0,BASE_NO 0,VB 100,VE 0,ACC 100,TRG_TIME 0,MOVE_TYPE #PTP_MOTION}
DECL E6POS P8={X 3086.77197,Y 287.191193,Z 1862.38,A -43.0205193,B 80.6090622,C -130.525208,S 2,T 11,E1 -1250.45398,E2 0.0,E3 0.0,E4 0.0,E5 0.0,E6 0.0}
DECL VW_MPARA_TYP P9_D={TOOL_NO 0,BASE_NO 0,VB 100,VE 0,ACC 100,TRG_TIME 0,MOVE_TYPE #PTP_MOTION}
DECL E6POS P9={X 3614.20093,Y -85.8147888,Z 1862.38,A -43.0205193,B 80.6090622,C -130.525208,S 2,T 10,E1 -1250.45398,E2 0.0,E3 0.0,E4 0.0,E5 0.0,E6 0.0}
DECL VW_MPARA_TYP P10_D={TOOL_NO 0,BASE_NO 0,VB 100,VE 0,ACC 100,TRG_TIME 0,MOVE_TYPE #PTP_MOTION}
DECL E6POS P10={X 2558.78198,Y -85.8147736,Z 1862.38,A -43.0205193,B 80.6090622,C -130.525208,S 2,T 10,E1 -1250.45398,E2 0.0,E3 0.0,E4 0.0,E5 0.0,E6 0.0}
DECL VW_MPARA_TYP P11_D={TOOL_NO 0,BASE_NO 0,VB 100,VE 0,ACC 100,TRG_TIME 0,MOVE_TYPE #PTP_MOTION}
DECL E6POS P11={X 2582.41797,Y 741.838623,Z 1862.38,A -43.0205193,B 80.6090622,C -130.525208,S 2,T 11,E1 -1250.45398,E2 0.0,E3 0.0,E4 0.0,E5 0.0,E6 0.0}
DECL VW_MPARA_TYP P12_D={TOOL_NO 0,BASE_NO 0,VB 100,VE 0,ACC 100,TRG_TIME 0,MOVE_TYPE #PTP_MOTION}
DECL E6POS P12={X 3679.87793,Y 664.384277,Z 1862.38,A -43.0205193,B 80.6090622,C -130.525208,S 2,T 11,E1 -1250.45398,E2 0.0,E3 0.0,E4 0.0,E5 0.0,E6 0.0}
DECL VW_MPARA_TYP P13_D={TOOL_NO 0,BASE_NO 0,VB 100,VE 0,ACC 100,TRG_TIME 0,MOVE_TYPE #PTP_MOTION}
DECL E6POS P13={X 890.547,Y 852.594421,Z 2209.01807,A 2.84489799,B 75.9217834,C -87.1302872,S 2,T 11,E1 -518.843,E2 0.0,E3 0.0,E4 0.0,E5 0.0,E6 0.0}
DECL VW_MPARA_TYP P14_D={TOOL_NO 0,BASE_NO 0,VB 100,VE 0,ACC 100,TRG_TIME 0,MOVE_TYPE #PTP_MOTION}
DECL E6POS P14={X 658.023376,Y 1250.53894,Z 1810.46399,A -20.2040405,B 74.9965515,C -110.919296,S 2,T 11,E1 -518.843,E2 0.0,E3 0.0,E4 0.0,E5 0.0,E6 0.0}
DECL VW_MPARA_TYP P15_D={TOOL_NO 21,BASE_NO 21,VB 100,VE 0,ACC 100,TRG_TIME 0,MOVE_TYPE #PTP_MOTION}
DECL E6POS P15={X -34.6645317,Y 154.178604,Z -0.000271785,A -110.204,B 74.9965515,C -110.919296,S 2,T 11,E1 -518.843,E2 0.0,E3 0.0,E4 0.0,E5 0.0,E6 0.0}
DECL VW_MPARA_TYP P16_D={TOOL_NO 21,BASE_NO 21,VB 100,VE 0,ACC 100,TRG_TIME 0,MOVE_TYPE #PTP_MOTION}
DECL E6POS P16={X -69.0514832,Y 226.887604,Z 214.548798,A -83.8805618,B 75.9134903,C -83.7540665,S 2,T 11,E1 -518.843323,E2 0.0,E3 0.0,E4 0.0,E5 0.0,E6 0.0}
DECL VW_MPARA_TYP P17_D={TOOL_NO 21,BASE_NO 21,VB 100,VE 0,ACC 100,TRG_TIME 0,MOVE_TYPE #PTP_MOTION}
DECL E6POS P17={X -22.3001595,Y 367.274109,Z 175.284103,A -81.3047485,B 75.8873367,C -81.0978165,S 2,T 11,E1 -518.843,E2 0.0,E3 0.0,E4 0.0,E5 0.0,E6 0.0}
DECL VW_MPARA_TYP P18_D={TOOL_NO 21,BASE_NO 21,VB 100,VE 0,ACC 100,TRG_TIME 0,MOVE_TYPE #PTP_MOTION}
DECL E6POS P18={X -22.2989597,Y 375.422913,Z 209.750198,A -81.3047485,B 75.8873367,C -81.0978165,S 2,T 11,E1 -518.843,E2 0.0,E3 0.0,E4 0.0,E5 0.0,E6 0.0}
DECL VW_MPARA_TYP P19_D={TOOL_NO 21,BASE_NO 21,VB 100,VE 0,ACC 100,TRG_TIME 0,MOVE_TYPE #PTP_MOTION}
DECL E6POS P19={X -13.4604702,Y 237.846603,Z 225.540207,A -81.3047485,B 75.8873367,C -81.0978165,S 2,T 11,E1 -518.843,E2 0.0,E3 0.0,E4 0.0,E5 0.0,E6 0.0}
DECL VW_MPARA_TYP P20_D={TOOL_NO 21,BASE_NO 21,VB 100,VE 0,ACC 100,TRG_TIME 0,MOVE_TYPE #PTP_MOTION}
DECL E6POS P20={X -13.7657204,Y 226.511597,Z 215.748505,A -81.3047485,B 75.8873367,C -81.0978165,S 2,T 11,E1 -518.843,E2 0.0,E3 0.0,E4 0.0,E5 0.0,E6 0.0}
DECL VW_MPARA_TYP P21_D={TOOL_NO 21,BASE_NO 21,VB 100,VE 0,ACC 100,TRG_TIME 0,MOVE_TYPE #PTP_MOTION}
DECL E6POS P21={X -16.0679893,Y -27.4565392,Z 246.361801,A -81.3069305,B 75.8837509,C -81.1000671,S 2,T 11,E1 -518.843,E2 0.0,E3 0.0,E4 0.0,E5 0.0,E6 0.0}
DECL VW_MPARA_TYP P22_D={TOOL_NO 21,BASE_NO 21,VB 100,VE 0,ACC 100,TRG_TIME 5,MOVE_TYPE #PTP_MOTION}
DECL E6POS P22={X -17.6393909,Y -38.4457207,Z 236.459900,A -81.3069305,B 75.8837509,C -81.1000671,S 2,T 11,E1 -518.843,E2 0.0,E3 0.0,E4 0.0,E5 0.0,E6 0.0}
DECL VW_MPARA_TYP P23_D={TOOL_NO 21,BASE_NO 21,VB 100,VE 0,ACC 100,TRG_TIME 0,MOVE_TYPE #PTP_MOTION}
DECL E6POS P23={X -33.9330101,Y -340.737915,Z 206.629196,A -81.3047485,B 75.8873367,C -81.0978165,S 2,T 11,E1 -518.843,E2 0.0,E3 0.0,E4 0.0,E5 0.0,E6 0.0}
DECL VW_MPARA_TYP P24_D={TOOL_NO 21,BASE_NO 21,VB 100,VE 0,ACC 100,TRG_TIME 0,MOVE_TYPE #PTP_MOTION}
DECL E6POS P24={X -27.1523304,Y -369.447388,Z 219.247803,A -81.3047485,B 75.8873367,C -81.0978165,S 2,T 11,E1 -518.843,E2 0.0,E3 0.0,E4 0.0,E5 0.0,E6 0.0}
DECL VW_MPARA_TYP P25_D={TOOL_NO 21,BASE_NO 21,VB 100,VE 0,ACC 100,TRG_TIME 0,MOVE_TYPE #PTP_MOTION}
DECL E6POS P25={X 16.4014702,Y 587.905884,Z -213.300903,A -67.1370773,B 76.4828491,C -83.5287628,S 2,T 11,E1 -518.843323,E2 0.0,E3 0.0,E4 0.0,E5 0.0,E6 0.0}
DECL VW_MPARA_TYP P26_D={TOOL_NO 21,BASE_NO 21,VB 100,VE 0,ACC 100,TRG_TIME 0,MOVE_TYPE #PTP_MOTION}
DECL E6POS P26={X -1.44520104,Y 541.245300,Z 126.166397,A -73.2554626,B 76.4828491,C -83.5287628,S 2,T 11,E1 -518.843323,E2 0.0,E3 0.0,E4 0.0,E5 0.0,E6 0.0}
DECL VW_MPARA_TYP P27_D={TOOL_NO 21,BASE_NO 21,VB 100,VE 0,ACC 100,TRG_TIME 0,MOVE_TYPE #PTP_MOTION}
DECL E6POS P27={X -869.461487,Y 274.278595,Z -626.534180,A 40.6801491,B -2.19141889,C -179.217606,S 2,T 11,E1 -518.843384,E2 0.0,E3 0.0,E4 0.0,E5 0.0,E6 0.0}
DECL VW_MPARA_TYP P28_D={TOOL_NO 21,BASE_NO 21,VB 100,VE 0,ACC 100,TRG_TIME 0,MOVE_TYPE #PTP_MOTION}
DECL E6POS P28={X -885.989197,Y -104.424,Z -595.999329,A 40.6801491,B -2.19141889,C -179.217606,S 2,T 11,E1 -518.843384,E2 0.0,E3 0.0,E4 0.0,E5 0.0,E6 0.0}
DECL VW_MPARA_TYP P29_D={TOOL_NO 21,BASE_NO 21,VB 100,VE 0,ACC 100,TRG_TIME 0,MOVE_TYPE #PTP_MOTION}
DECL E6POS P29={X -917.093872,Y -413.263885,Z -576.676575,A 33.4063911,B -2.19141889,C -179.217606,S 2,T 11,E1 -518.843384,E2 0.0,E3 0.0,E4 0.0,E5 0.0,E6 0.0}
DECL VW_MPARA_TYP P30_D={TOOL_NO 21,BASE_NO 21,VB 100,VE 0,ACC 100,TRG_TIME 0,MOVE_TYPE #PTP_MOTION}
DECL E6POS P30={X -857.319702,Y 426.212891,Z -1065.24500,A 44.0755692,B -2.72070098,C -178.624802,S 2,T 11,E1 -518.843384,E2 0.0,E3 0.0,E4 0.0,E5 0.0,E6 0.0}
DECL VW_MPARA_TYP P31_D={TOOL_NO 0,BASE_NO 0,VB 100,VE 0,ACC 100,TRG_TIME 0,MOVE_TYPE #PTP_MOTION}
DECL E6POS P31={X 466.588898,Y 1714.05188,Z 1641.94983,A 93.1114273,B -2.11931801,C -179.406097,S 2,T 11,E1 -518.843384,E2 0.0,E3 0.0,E4 0.0,E5 0.0,E6 0.0}
ENDDAT
